Yaskawa INFORM job: R1_72,2(0,0)KM-OK.JBI

/JOB
//NAME R1_72,2(0,0)KM-OK
///FOLDERNAME KRIS-SCIANA
//POS
///NPOS 76,76,0,3,0,0
///TOOL 0
///POSTYPE PULSE
///PULSE
C00000=214739,-34142,-86579,18171,90882,-33584
C00001=192628,-9219,-68940,27221,97535,-38774
C00002=192628,-9219,-68940,27221,97535,-38774
C00003=206785,1928,-2866,24835,77749,-31705
C00004=211412,-5691,-9151,24019,76339,-30254
C00005=211721,-3296,-4468,24119,74735,-30470
C00006=211721,-2988,-3159,24186,74143,-30595
C00007=211721,-3286,-4423,24121,74715,-30475
C00008=212044,-1475,-2934,24060,74632,-30369
C00009=211721,-3286,-4423,24121,74715,-30475
C00010=204612,2210,-14410,24827,85008,-30989
C00011=204612,18022,-42675,26555,108188,-25943
C00012=214739,-34142,-86579,18171,90882,-33584
C00013=216406,-37850,-86218,17444,88554,-33440
C00014=217080,-39257,-86022,17157,87628,-33372
C00015=216891,-43789,-85751,17261,85277,-33761
C00016=217262,-41380,-84303,17098,85542,-33611
C00017=217436,-41971,-84662,17026,85428,-33572
C00018=217080,-39257,-86022,17157,87628,-33372
C00019=216120,-38690,-85533,17566,87791,-33633
C00020=216269,-39865,-84982,17508,86862,-33722
C00021=216120,-38690,-85533,17566,87791,-33633
C00022=217080,-39257,-86022,17157,87628,-33372
C00023=201345,-20375,-78021,31054,112530,-39584
C00024=201639,-23474,-77107,30489,110579,-40057
C00025=202590,-24455,-77954,30278,110316,-39807
C00026=201639,-23474,-77107,30489,110579,-40057
C00027=201345,-20375,-78021,31054,112530,-39584
C00028=205311,-24199,-81401,30131,111496,-38553
C00029=204414,-22055,-81146,30572,112570,-38540
C00030=202220,-16510,-80317,31730,115203,-38470
C00031=184984,-3292,-66527,21578,97839,-52041
C00032=187848,106335,29423,-5768,95800,74791
C00033=187846,93398,30248,-5715,88678,75115
C00034=187845,90841,31211,-5716,86781,75201
C00035=186749,80935,25217,37882,97144,45469
C00036=188249,88132,29282,-5868,86603,75331
C00037=187781,90810,31570,-5693,86541,75193
C00038=186593,79700,23961,37938,97314,45468
C00039=186285,79829,24181,38011,97380,45375
C00040=186155,80197,24595,38034,97381,45324
C00041=185994,80326,25273,38042,97165,45186
C00042=185838,79602,22632,38213,98224,45505
C00043=185327,80011,19037,38655,100344,46081
C00044=124459,133068,90612,6691,115644,64898
C00045=124459,133068,90612,6691,115644,64898
C00046=93275,113796,34371,-3502,120109,70620
C00047=89315,113601,52844,2619,120646,72485
C00048=89316,111310,53557,2572,119031,72446
C00049=89697,121055,69415,651,117839,72105
C00050=89348,111517,54075,2569,118818,72453
C00051=89564,113087,57614,2554,117442,72498
C00052=90033,119920,67876,706,118200,72231
C00053=91337,116538,63361,923,119232,72724
C00054=99842,93639,33750,-17614,115849,72169
C00055=99880,92745,32649,-17651,116064,72149
C00056=99324,86551,24395,-17976,117766,71666
C00057=94613,96171,29214,-8772,122473,71759
C00058=95513,127998,72000,-2391,121454,32503
C00059=95373,128312,72443,-2414,81128,32453
C00060=95373,169527,125925,-4488,33256,32455
C00061=126436,146554,76460,6599,53537,-23923
C00062=95373,169524,125926,-4503,33256,32457
C00063=142575,-91178,-115388,39866,103652,-54544
C00064=192628,-9219,-68940,27221,97535,-38774
C00065=206785,1928,-2866,24835,77749,-31705
C00066=209029,-3383,-7279,24450,77069,-31002
C00067=209515,-206,-2001,24513,75448,-31160
C00068=211877,3032,462,21685,76563,-30091
C00069=215265,-130,-2171,21101,75678,-28996
C00070=214513,-2176,-4685,21195,76334,-29157
C00071=209029,-3383,-7279,24450,77069,-31002
C00072=192628,-9219,-68940,27221,97535,-38774
C00073=135854,-98188,-118079,40471,104995,-56824
C00074=123760,23071,-66067,30293,113844,-22684
C00075=95373,169527,125925,-4488,33256,32455
BC00000=352013,15,1075175
BC00001=352013,15,1075175
BC00002=365574,15,642260
BC00003=365574,15,642260
BC00004=365574,15,642260
BC00005=365574,15,642260
BC00006=365574,15,642260
BC00007=365574,15,642260
BC00008=365574,15,642260
BC00009=365574,15,642260
BC00010=365574,15,642260
BC00011=365574,15,1075175
BC00012=352013,15,1075175
BC00013=346494,15,1075175
BC00014=344287,15,1075175
BC00015=341901,15,1075175
BC00016=341901,15,1075175
BC00017=344290,15,1075175
BC00018=344287,15,1075175
BC00019=338131,15,1075175
BC00020=338132,15,1075175
BC00021=338131,15,1075175
BC00022=344287,15,1075175
BC00023=302697,15,1075175
BC00024=302700,15,1075175
BC00025=302719,15,1075175
BC00026=302700,15,1075175
BC00027=302697,15,1075175
BC00028=316402,15,1075175
BC00029=317723,15,1075175
BC00030=321027,15,1075175
BC00031=333173,81717,1075175
BC00032=376146,194177,1075175
BC00033=376146,194177,1075175
BC00034=376277,192427,1075175
BC00035=398174,122098,1075175
BC00036=376329,191727,1075175
BC00037=376329,191727,1075175
BC00038=398174,122098,1075175
BC00039=398174,122098,1075175
BC00040=398174,122098,1075175
BC00041=398174,116514,1075175
BC00042=398174,116400,1075175
BC00043=398174,116114,1075175
BC00044=235371,182236,1075175
BC00045=16839,182236,1075175
BC00046=13012,209674,1075175
BC00047=13012,209674,1075175
BC00048=13735,213189,1075175
BC00049=14024,214595,1075175
BC00050=14024,214595,1075175
BC00051=14024,214595,1075175
BC00052=14024,214595,1075175
BC00053=14024,214595,1075175
BC00054=14024,214595,1075175
BC00055=14024,214595,1075175
BC00056=14024,214595,1075175
BC00057=14024,214595,1075175
BC00058=10344,234287,1075175
BC00059=10344,234287,1075175
BC00060=10345,234286,1075173
BC00061=262155,152897,1075174
BC00062=327786,234286,1075172
BC00063=352013,111996,1075175
BC00064=352013,15,1075175
BC00065=365574,15,642260
BC00066=365574,15,642260
BC00067=365574,15,642260
BC00068=365574,15,642260
BC00069=365574,15,642260
BC00070=365574,15,642260
BC00071=365574,15,642260
BC00072=352013,15,1075175
BC00073=352013,397246,1075175
BC00074=249935,462030,1075174
BC00075=10345,614086,1075173
///POSTYPE BASE
///RECTAN
///RCONF 0,0,0,0,1,0,0,0,0,0,0,0,0,0,0,0,0,0,0,0,0,0,0,0
P00006=2.006,1.622,-0.565,0.0000,0.0000,0.0000
P00021=0.073,2.058,-0.109,0.0000,0.0000,0.0000
///RCONF 0,0,0,0,0,0,0,0,0,0,0,0,0,0,0,0,0,0,0,0,0,0,0,0
P00030=-0.014,-0.768,0.131,0.0000,0.0000,0.0000
//INST
///DATE 2024/09/16 12:16
///ATTR SC,RW
///GROUP1 RB1,BS1
NOP
'R1_72.2(0,0)
'Path S1563
SFTOF
MOVJ C00000 BC00000 VJ=70.00
MOVJ C00001 BC00001 VJ=70.00
MOVJ C00002 BC00002 VJ=70.00
MOVJ C00003 BC00003 VJ=70.00
MOVL C00004 BC00004 V=166.7
MOVL C00005 BC00005 V=100.0
REFP 3 C00006 BC00006
CALL JOB:SEARCH-R1
SET P030 P006
SFTON P030
MOVL C00007 BC00007 V=100.0
REFP 3 C00008 BC00008
CALL JOB:SEARCH-R1
SET P030 P006
SFTON P030
MOVL C00009 BC00009 V=100.0
SFTOF
MOVL C00010 BC00010 V=400.0
MOVL C00011 BC00011 V=1000.0
MOVJ C00012 BC00012 VJ=70.00
MOVJ C00013 BC00013 VJ=50.00
MOVL C00014 BC00014 V=100.0
MOVL C00015 BC00015 V=60.0
REFP 3 C00016 BC00016
CALL JOB:SEARCH-R1
SET P021 P006
SFTON P021
MOVL C00017 BC00017 V=60.0
MOVL C00018 BC00018 V=100.0
MOVL C00019 BC00019 V=60.0
REFP 3 C00020 BC00020
CALL JOB:SEARCH-R1
SET P021 P006
SFTON P021
MOVL C00021 BC00021 V=60.0
MOVL C00022 BC00022 V=100.0
MOVL C00023 BC00023 V=100.0
MOVL C00024 BC00024 V=60.0
REFP 3 C00025 BC00025
CALL JOB:SEARCH-R1
SET P021 P006
SFTON P021
MOVL C00026 BC00026 V=60.0
MOVL C00027 BC00027 V=100.0
MOVL C00028 BC00028 V=100.0
MOVL C00029 BC00029 V=166.7
MOVL C00030 BC00030 V=166.7
'Path VIA1564
SFTOF
MOVJ C00031 BC00031 VJ=50.00
'Path W1561
SFTOF
SFTON P021
CALL JOB:COFNIJ_DRUT
MOVJ C00032 BC00032 VJ=50.00
MOVJ C00033 BC00033 VJ=100.00
MOVJ C00034 BC00034 VJ=100.00
MOVL C00035 BC00035 V=166.7 PL=0
REFP 1 C00036 BC00036
REFP 2 C00037 BC00037
MACRO1 MJ#(0) ARGF6
ARCON
MOVL C00038 BC00038 V=10.8
MOVL C00039 BC00039 V=10.8
MOVL C00040 BC00040 V=10.8
MOVL C00041 BC00041 V=10.8
ARCOF
MOVL C00042 BC00042 V=100.0
MOVL C00043 BC00043 V=166.7
SFTOF
'Path VIA1565
SFTOF
MOVJ C00044 BC00044 VJ=50.00
MOVJ C00045 BC00045 VJ=50.00
'Path W1566
SFTOF
SFTON P021
MOVJ C00046 BC00046 VJ=100.00
MOVJ C00047 BC00047 VJ=100.00
MOVJ C00048 BC00048 VJ=50.00
MOVL C00049 BC00049 V=100.0 PL=0
REFP 1 C00050 BC00050
REFP 2 C00051 BC00051
MACRO1 MJ#(0) ARGF5
ARCON
MOVL C00052 BC00052 V=8.3
MOVL C00053 BC00053 V=8.3
ARCOF
MOVL C00054 BC00054 V=10.0
ARCON
MOVL C00055 BC00055 V=8.3
MOVL C00056 BC00056 V=8.3
ARCOF
MOVL C00057 BC00057 V=166.7
MOVL C00058 BC00058 V=166.7
SFTOF
MOVJ C00059 BC00059 VJ=50.00
MOVJ C00060 BC00060 VJ=100.00
MOVJ C00061 BC00061 VJ=70.00
MOVL C00062 BC00062 V=1000.0
MOVJ C00063 BC00063 VJ=70.00
MOVJ C00064 BC00064 VJ=70.00
MOVJ C00065 BC00065 VJ=70.00
MOVL C00066 BC00066 V=166.7
SFTON P030
MOVL C00067 BC00067 V=100.0
MOVL C00068 BC00068 V=100.0 PL=0
MACRO1 MJ#(0) ARGF7
ARCON
MOVL C00069 BC00069 V=9.2
ARCOF
MOVL C00070 BC00070 V=233.3
SFTOF
MOVL C00071 BC00071 V=333.3
MOVL C00072 BC00072 V=666.7
MOVJ C00073 BC00073 VJ=70.00
MOVJ C00074 BC00074 VJ=70.00
MOVJ C00075 BC00075 VJ=100.00
END
